FUNCTION_BLOCK FB_Handle_Emergency
VAR_INPUT
    execute: 				BOOL;
END_VAR
VAR_OUTPUT
    busy: 					BOOL;
END_VAR
VAR
    state: 					INT := 0;
    tonDelay: 				TON;
	
	allActionsCompleteShutdown:		BOOL;
	RecoveryToMaintenance:							BOOL;
END_VAR

//What is happening here?
IF execute <> TRUE THEN
	
    state := 0;
    busy := FALSE;
    tonDelay(IN := FALSE);
	
    RETURN;
END_IF

busy := TRUE;

CASE state OF
	
    0:  GVL_FSM.b_EmergencyLine := FALSE;
		
        GVL_Prop.propulsion_enable := FALSE;
        GVL_LEVI.levitation_enable := FALSE;
		
        state := 1;
        
    1:	allActionsCompleteShutdown := NOT GVL_LEVI.levitation_active 
		AND NOT GVL_Prop.propulsion_active 
		AND GVL_Levi.DC_LINK_SAFE 
		AND GVL_Prop.DC_LINK_SAFE 
		AND GVL_FSM.bbrakes_engaged; 
	
        IF allActionsCompleteShutdown THEN
			
			  state := 2;
		
        END_IF
		
    2:	RecoveryToMaintenance := 
	
		NOT GVL_Prop.propulsion_fault AND
		NOT GVL_LEVI.levitation_fault AND
		
		BasicChecks() AND 
		
		NOT GVL_THERMAL.bMOTOROVERHEAT AND 
		NOT GVL_THERMAL.bHEMSOVERHEAT AND
		NOT GVL_THERMAL.bEMSOVERHEAT AND
		NOT GVL_THERMAL.bFLOWOVERHEAT;
		
		IF RecoveryToMaintenance THEN
			
			GVL_FSM.b_EmergencyLine := TRUE;
			
			state := 3;
			
		END_IF
	//not sure if we dont get the same error with the brakes and SDC resetting that we go into a maintenance to emergency loop. Since the maintenance command is explciti the FSM might have time to reset.
		    
    3:	tonDelay(IN := TRUE, PT := T#2S);
        IF tonDelay.Q AND GVL_FSM.bsdc_closed THEN
			
            busy := FALSE;
			execute := FALSE;
			state := 0;
			tonDelay(IN := FALSE);
        END_IF
END_CASE

END_FUNCTION_BLOCK

(* stored: Version 1.1.0.1
   POU FB_Handle_Emergency: Id {5e0fb178-c06f-42de-8ba0-d84d3592dd6b}, SpecialFunc None *)
